# EPICS autosave request: iocBoot/sioc-asta-lake01/lakeshore336.req
file ../lakeshoreCommon.req P=$(P)
